(*
Searches an `I_Entity` for a `I_Tag` component with provided `Option` value.
Result:
- Ok - Returns iTag.
- None - Returns null.
- Err.Itf0 - Returns null, incorrect interface.
*)
FUNCTION GetTagOpt : Result
VAR_INPUT
	iEntity		: I_Entity;
	sOption		: Str;
END_VAR
VAR_OUTPUT
	iTag		: I_Tag;
END_VAR
VAR
	i			: Iter(1);
	_iComp		: I_FatComponent;
END_VAR

IF iEntity = 0 THEN
	GetTagOpt := Err.Itf0;
	RETURN;
END_IF

WHILE IsOk(iEntity.Get(i.Next(), iComp => _iComp)) DO
	IF IsOk(ICompToITag(_iComp.Raw, iDest => iTag)) THEN
		IF iTag.Option = sOption THEN
			GetTagOpt := Ok;
			RETURN;
		ELSE
			iTag := 0;
		END_IF
	END_IF
END_WHILE

END_FUNCTION

(* stored: Version 1.1.0.1
   POU GetTagOpt: Id {b48ed172-a791-460c-b58e-fd210c4dcaad}, SpecialFunc None *)
